INTERFACE IDisplay EXTENDS IBase

METHOD Show : BOOL
VAR_INPUT
	Message : T_MaxString;
END_VAR
END_METHOD

END_INTERFACE

(* stored: Version 1.1.0.1, ProductVersion 3.1.4024.12
   Itf IDisplay: Id {c20bdbc7-b695-4a99-bf2b-941ddf6b7391}
   Method Show: Id {127aacfe-754b-4c6f-876f-57be1f081f52} *)
